{attribute 'qualified_only'}
//{attribute 'strict'}
TYPE ConveyorMode :
(
	IDLE,
	FORWARD,
	BACKWARD,
	STOP,
	
	size
);
END_TYPE

(* stored: Version 1.1.0.1, ProductVersion 3.1.4024.11
   DUT ConveyorMode: Id {f3ae7e6a-94c4-464b-b92e-c21b5e4f5c85} *)
